FUNCTION CharIsNumberOrPeriod : BOOL
VAR_INPUT
   bChar : BYTE; // char to check
END_VAR

// check is bChar in number range of ascii, or a period (full-stop).
CharIsNumberOrPeriod := CharIsNumber(bChar) OR_ELSE (bChar = 46);

END_FUNCTION

(* stored: Version 1.1.0.1, ProductVersion 3.1.4024.9
   POU CharIsNumberOrPeriod: Id {3d88a1e5-09f2-473b-9457-e0e61ca45782}, SpecialFunc None *)
